Staubli VAL3: AXISMOVER.dtx

public string sItems
public bool bAxisMove
